PROGRAM MAIN
VAR
	ConfigRoot : FB_ConfigRoot;
END_VAR

Run(ApplicationConfigRoot := ConfigRoot);

END_PROGRAM

(* stored: Version 1.1.0.1, ProductVersion 3.1.4026.18
   POU MAIN: Id {732eef67-564b-4eae-a87a-e2bb58901008}, SpecialFunc None *)
